// TIA Portal V17 export
// export: Created 2025-03-07T09:17:58.1405762Z, ExportSetting WithDefaults, DisplayName Totally Integrated Automation Portal, DisplayVersion V17 Update 8, DisplayName TIA Portal Openness, DisplayVersion V17 Update 8, DisplayName TIA Portal Version Control Interface, DisplayVersion V17, DisplayName SINAMICS Startdrive Advanced, DisplayVersion V17 SP2, DisplayName SINAMICS Startdrive G110M, G120, G120C, G120D, G120P, G115D, DisplayVersion V17 SP2, DisplayName SINAMICS Startdrive G130, G150, S120, S150, SINAMICS MV, S210, DisplayVersion V17 SP2, DisplayName STEP 7 Professional, DisplayVersion V17 Update 8, DisplayName SINUMERIK ONE STEP 7 Toolbox, DisplayVersion V17 Update 12, DisplayName SINUMERIK 840D sl STEP 7 Toolbox, DisplayVersion V17 Update 12, DisplayName STEP 7 Safety, DisplayVersion V17 Update 6, DisplayName WinCC Advanced, DisplayVersion V17 Update 8
FUNCTION "FC1213_HOME_UNIT_01_STATION_1" : Void   // FC1213, LAD
{ S7_Optimized_Access := 'FALSE' }
AUTHOR : ETXETAR
VERSION : 1.0
// stored: AutoNumber false, IsIECCheckEnabled false, SetENOAutomatically false, UDAEnableTagReadback false
   VAR_TEMP
      UNIT_01_STATION_1_LOCAL_E_RETURNS : Bool;   // UNIT 01 STATION 1 LOCAL E RETURNS
      UNIT_01_STATION_1_MACHINE_E_RETURNS : Bool;   // UNIT 01 STATION 1 MACHINE E RETURNS
   END_VAR
   VAR CONSTANT
      FC_NUMBER : DInt := 1213;
   END_VAR
   VAR_TEMP   // added for the SCL form of the ladder/FBD networks
      _w1 : Bool;
      _w2 : Bool;
   END_VAR
BEGIN

REGION Network 1: GENERAL CONDITIONS
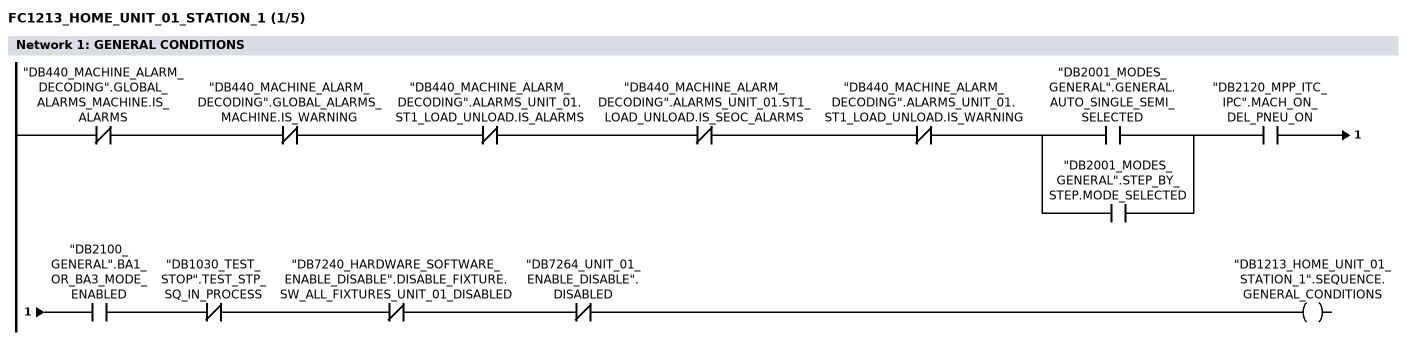
   RUNG wire#powerrail
      I_Contact( "DB440_MACHINE_ALARM_DECODING".GLOBAL_ALARMS_MACHINE.IS_ALARMS )
      I_Contact( "DB440_MACHINE_ALARM_DECODING".GLOBAL_ALARMS_MACHINE.IS_WARNING )
      I_Contact( "DB440_MACHINE_ALARM_DECODING".ALARMS_UNIT_01.ST1_LOAD_UNLOAD.IS_ALARMS )
      I_Contact( "DB440_MACHINE_ALARM_DECODING".ALARMS_UNIT_01.ST1_LOAD_UNLOAD.IS_SEOC_ALARMS )
      I_Contact( "DB440_MACHINE_ALARM_DECODING".ALARMS_UNIT_01.ST1_LOAD_UNLOAD.IS_WARNING )
      wire#w1
      Contact( "DB2001_MODES_GENERAL".GENERAL.AUTO_SINGLE_SEMI_SELECTED )
      wire#w2
      Contact( "DB2120_MPP_ITC_IPC".MACH_ON_DEL_PNEU_ON )
      Contact( "DB2100_GENERAL".BA1_OR_BA3_MODE_ENABLED )
      I_Contact( "DB1030_TEST_STOP".TEST_STP_SQ_IN_PROCESS )
      I_Contact( "DB7240_HARDWARE_SOFTWARE_ENABLE_DISABLE".DISABLE_FIXTURE.SW_ALL_FIXTURES_UNIT_01_DISABLED )
      I_Contact( "DB7264_UNIT_01_ENABLE_DISABLE".DISABLED )
      Coil( "DB1213_HOME_UNIT_01_STATION_1".SEQUENCE.GENERAL_CONDITIONS )
   END_RUNG
   RUNG wire#w1
      Contact( "DB2001_MODES_GENERAL".STEP_BY_STEP.MODE_SELECTED )
   END_RUNG wire#w2
   // the same network as SCL:
   "DB1213_HOME_UNIT_01_STATION_1".SEQUENCE.GENERAL_CONDITIONS := NOT "DB440_MACHINE_ALARM_DECODING".GLOBAL_ALARMS_MACHINE.IS_ALARMS AND NOT "DB440_MACHINE_ALARM_DECODING".GLOBAL_ALARMS_MACHINE.IS_WARNING AND NOT "DB440_MACHINE_ALARM_DECODING".ALARMS_UNIT_01.ST1_LOAD_UNLOAD.IS_ALARMS AND NOT "DB440_MACHINE_ALARM_DECODING".ALARMS_UNIT_01.ST1_LOAD_UNLOAD.IS_SEOC_ALARMS AND NOT "DB440_MACHINE_ALARM_DECODING".ALARMS_UNIT_01.ST1_LOAD_UNLOAD.IS_WARNING AND ("DB2001_MODES_GENERAL".GENERAL.AUTO_SINGLE_SEMI_SELECTED OR "DB2001_MODES_GENERAL".STEP_BY_STEP.MODE_SELECTED) AND "DB2120_MPP_ITC_IPC".MACH_ON_DEL_PNEU_ON AND "DB2100_GENERAL".BA1_OR_BA3_MODE_ENABLED AND NOT "DB1030_TEST_STOP".TEST_STP_SQ_IN_PROCESS AND NOT "DB7240_HARDWARE_SOFTWARE_ENABLE_DISABLE".DISABLE_FIXTURE.SW_ALL_FIXTURES_UNIT_01_DISABLED AND NOT "DB7264_UNIT_01_ENABLE_DISABLE".DISABLED;
END_REGION

REGION Network 2: OPERATOR HELP
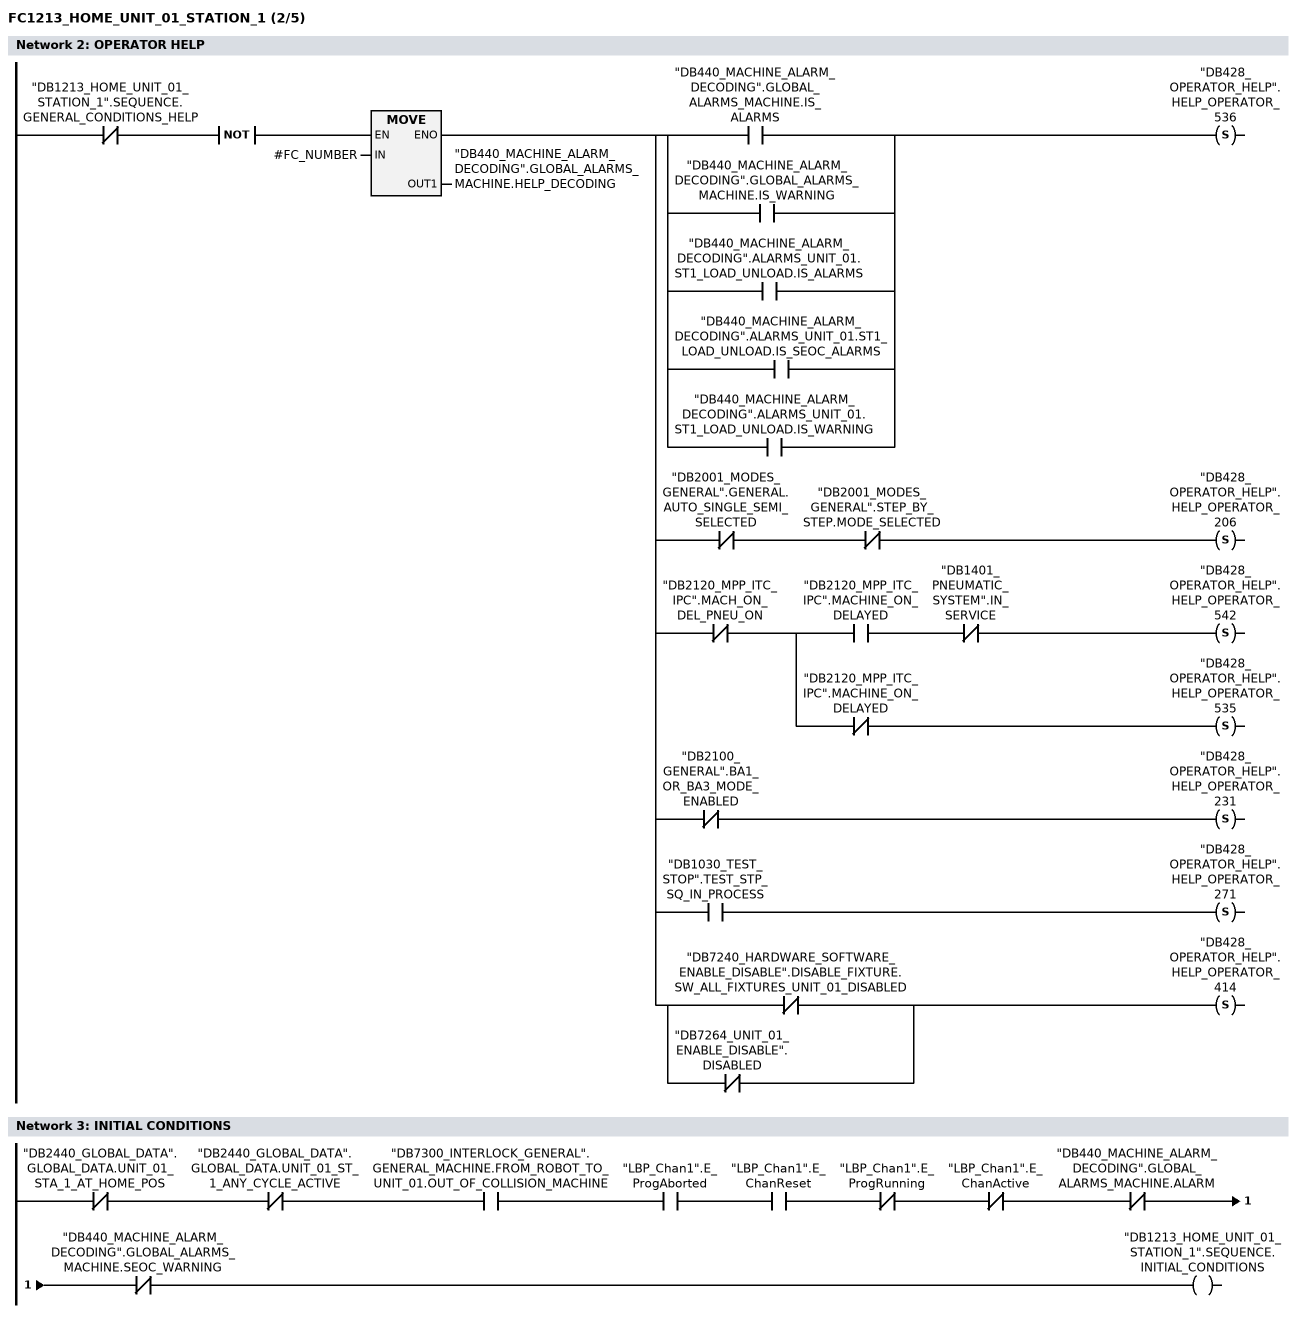
   RUNG wire#powerrail
      I_Contact( "DB1213_HOME_UNIT_01_STATION_1".SEQUENCE.GENERAL_CONDITIONS_HELP )
      Not()
      { S7_GenerateENO := "TRUE" } Move(in := #FC_NUMBER, out1 => "DB440_MACHINE_ALARM_DECODING".GLOBAL_ALARMS_MACHINE.HELP_DECODING)
      wire#w1
      Contact( "DB440_MACHINE_ALARM_DECODING".GLOBAL_ALARMS_MACHINE.IS_ALARMS )
      wire#w2
      S_Coil( "DB428_OPERATOR_HELP".HELP_OPERATOR_536 )
   END_RUNG
   RUNG wire#w1
      Contact( "DB440_MACHINE_ALARM_DECODING".GLOBAL_ALARMS_MACHINE.IS_WARNING )
   END_RUNG wire#w2
   RUNG wire#w1
      Contact( "DB440_MACHINE_ALARM_DECODING".ALARMS_UNIT_01.ST1_LOAD_UNLOAD.IS_ALARMS )
   END_RUNG wire#w2
   RUNG wire#w1
      Contact( "DB440_MACHINE_ALARM_DECODING".ALARMS_UNIT_01.ST1_LOAD_UNLOAD.IS_SEOC_ALARMS )
   END_RUNG wire#w2
   RUNG wire#w1
      Contact( "DB440_MACHINE_ALARM_DECODING".ALARMS_UNIT_01.ST1_LOAD_UNLOAD.IS_WARNING )
   END_RUNG wire#w2
   RUNG wire#w1
      I_Contact( "DB2001_MODES_GENERAL".GENERAL.AUTO_SINGLE_SEMI_SELECTED )
      I_Contact( "DB2001_MODES_GENERAL".STEP_BY_STEP.MODE_SELECTED )
      S_Coil( "DB428_OPERATOR_HELP".HELP_OPERATOR_206 )
   END_RUNG
   RUNG wire#w1
      I_Contact( "DB2120_MPP_ITC_IPC".MACH_ON_DEL_PNEU_ON )
      wire#w3
      Contact( "DB2120_MPP_ITC_IPC".MACHINE_ON_DELAYED )
      I_Contact( "DB1401_PNEUMATIC_SYSTEM".IN_SERVICE )
      S_Coil( "DB428_OPERATOR_HELP".HELP_OPERATOR_542 )
   END_RUNG
   RUNG wire#w3
      I_Contact( "DB2120_MPP_ITC_IPC".MACHINE_ON_DELAYED )
      S_Coil( "DB428_OPERATOR_HELP".HELP_OPERATOR_535 )
   END_RUNG
   RUNG wire#w1
      I_Contact( "DB2100_GENERAL".BA1_OR_BA3_MODE_ENABLED )
      S_Coil( "DB428_OPERATOR_HELP".HELP_OPERATOR_231 )
   END_RUNG
   RUNG wire#w1
      Contact( "DB1030_TEST_STOP".TEST_STP_SQ_IN_PROCESS )
      S_Coil( "DB428_OPERATOR_HELP".HELP_OPERATOR_271 )
   END_RUNG
   RUNG wire#w1
      I_Contact( "DB7240_HARDWARE_SOFTWARE_ENABLE_DISABLE".DISABLE_FIXTURE.SW_ALL_FIXTURES_UNIT_01_DISABLED )
      wire#w4
      S_Coil( "DB428_OPERATOR_HELP".HELP_OPERATOR_414 )
   END_RUNG
   RUNG wire#w1
      I_Contact( "DB7264_UNIT_01_ENABLE_DISABLE".DISABLED )
   END_RUNG wire#w4
   // the same network as SCL:
   // ENO of a box is taken as its EN; it also drops when the box reports an error
   #_w1 := NOT (NOT "DB1213_HOME_UNIT_01_STATION_1".SEQUENCE.GENERAL_CONDITIONS_HELP);
   IF #_w1 THEN "DB440_MACHINE_ALARM_DECODING".GLOBAL_ALARMS_MACHINE.HELP_DECODING := #FC_NUMBER; END_IF;
   IF #_w1 AND ("DB440_MACHINE_ALARM_DECODING".GLOBAL_ALARMS_MACHINE.IS_ALARMS OR "DB440_MACHINE_ALARM_DECODING".GLOBAL_ALARMS_MACHINE.IS_WARNING OR "DB440_MACHINE_ALARM_DECODING".ALARMS_UNIT_01.ST1_LOAD_UNLOAD.IS_ALARMS OR "DB440_MACHINE_ALARM_DECODING".ALARMS_UNIT_01.ST1_LOAD_UNLOAD.IS_SEOC_ALARMS OR "DB440_MACHINE_ALARM_DECODING".ALARMS_UNIT_01.ST1_LOAD_UNLOAD.IS_WARNING) THEN
       "DB428_OPERATOR_HELP".HELP_OPERATOR_536 := TRUE;
   END_IF;
   IF #_w1 AND NOT "DB2001_MODES_GENERAL".GENERAL.AUTO_SINGLE_SEMI_SELECTED AND NOT "DB2001_MODES_GENERAL".STEP_BY_STEP.MODE_SELECTED THEN
       "DB428_OPERATOR_HELP".HELP_OPERATOR_206 := TRUE;
   END_IF;
   #_w2 := #_w1 AND NOT "DB2120_MPP_ITC_IPC".MACH_ON_DEL_PNEU_ON;
   IF #_w2 AND "DB2120_MPP_ITC_IPC".MACHINE_ON_DELAYED AND NOT "DB1401_PNEUMATIC_SYSTEM".IN_SERVICE THEN
       "DB428_OPERATOR_HELP".HELP_OPERATOR_542 := TRUE;
   END_IF;
   IF #_w2 AND NOT "DB2120_MPP_ITC_IPC".MACHINE_ON_DELAYED THEN
       "DB428_OPERATOR_HELP".HELP_OPERATOR_535 := TRUE;
   END_IF;
   IF #_w1 AND NOT "DB2100_GENERAL".BA1_OR_BA3_MODE_ENABLED THEN
       "DB428_OPERATOR_HELP".HELP_OPERATOR_231 := TRUE;
   END_IF;
   IF #_w1 AND "DB1030_TEST_STOP".TEST_STP_SQ_IN_PROCESS THEN
       "DB428_OPERATOR_HELP".HELP_OPERATOR_271 := TRUE;
   END_IF;
   IF #_w1 AND (NOT "DB7240_HARDWARE_SOFTWARE_ENABLE_DISABLE".DISABLE_FIXTURE.SW_ALL_FIXTURES_UNIT_01_DISABLED OR NOT "DB7264_UNIT_01_ENABLE_DISABLE".DISABLED) THEN
       "DB428_OPERATOR_HELP".HELP_OPERATOR_414 := TRUE;
   END_IF;
END_REGION

REGION Network 3: INITIAL CONDITIONS
   RUNG wire#powerrail
      I_Contact( "DB2440_GLOBAL_DATA".GLOBAL_DATA.UNIT_01_STA_1_AT_HOME_POS )
      I_Contact( "DB2440_GLOBAL_DATA".GLOBAL_DATA.UNIT_01_ST_1_ANY_CYCLE_ACTIVE )
      Contact( "DB7300_INTERLOCK_GENERAL".GENERAL_MACHINE.FROM_ROBOT_TO_UNIT_01.OUT_OF_COLLISION_MACHINE )
      Contact( "LBP_Chan1".E_ProgAborted )
      Contact( "LBP_Chan1".E_ChanReset )
      I_Contact( "LBP_Chan1".E_ProgRunning )
      I_Contact( "LBP_Chan1".E_ChanActive )
      I_Contact( "DB440_MACHINE_ALARM_DECODING".GLOBAL_ALARMS_MACHINE.ALARM )
      I_Contact( "DB440_MACHINE_ALARM_DECODING".GLOBAL_ALARMS_MACHINE.SEOC_WARNING )
      Coil( "DB1213_HOME_UNIT_01_STATION_1".SEQUENCE.INITIAL_CONDITIONS )
   END_RUNG
   // the same network as SCL:
   "DB1213_HOME_UNIT_01_STATION_1".SEQUENCE.INITIAL_CONDITIONS := NOT "DB2440_GLOBAL_DATA".GLOBAL_DATA.UNIT_01_STA_1_AT_HOME_POS AND NOT "DB2440_GLOBAL_DATA".GLOBAL_DATA.UNIT_01_ST_1_ANY_CYCLE_ACTIVE AND "DB7300_INTERLOCK_GENERAL".GENERAL_MACHINE.FROM_ROBOT_TO_UNIT_01.OUT_OF_COLLISION_MACHINE AND "LBP_Chan1".E_ProgAborted AND "LBP_Chan1".E_ChanReset AND NOT "LBP_Chan1".E_ProgRunning AND NOT "LBP_Chan1".E_ChanActive AND NOT "DB440_MACHINE_ALARM_DECODING".GLOBAL_ALARMS_MACHINE.ALARM AND NOT "DB440_MACHINE_ALARM_DECODING".GLOBAL_ALARMS_MACHINE.SEOC_WARNING;
END_REGION

REGION Network 4: OPERATOR HELP
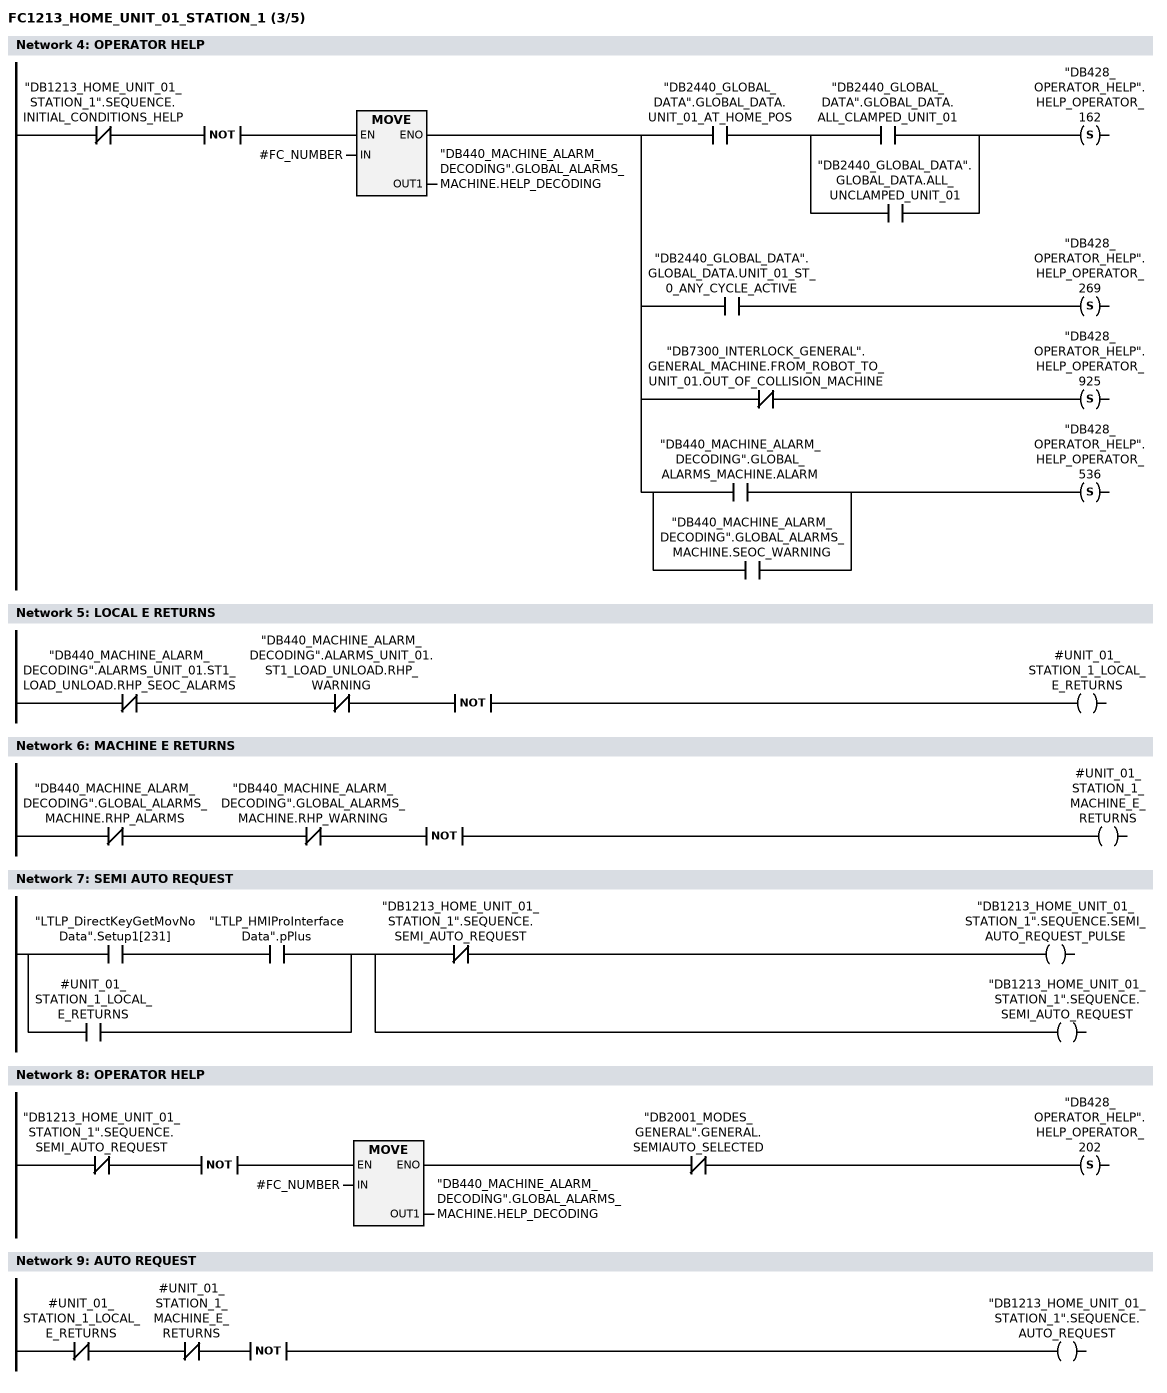
   RUNG wire#powerrail
      I_Contact( "DB1213_HOME_UNIT_01_STATION_1".SEQUENCE.INITIAL_CONDITIONS_HELP )
      Not()
      { S7_GenerateENO := "TRUE" } Move(in := #FC_NUMBER, out1 => "DB440_MACHINE_ALARM_DECODING".GLOBAL_ALARMS_MACHINE.HELP_DECODING)
      wire#w1
      Contact( "DB2440_GLOBAL_DATA".GLOBAL_DATA.UNIT_01_AT_HOME_POS )
      wire#w2
      Contact( "DB2440_GLOBAL_DATA".GLOBAL_DATA.ALL_CLAMPED_UNIT_01 )
      wire#w3
      S_Coil( "DB428_OPERATOR_HELP".HELP_OPERATOR_162 )
   END_RUNG
   RUNG wire#w2
      Contact( "DB2440_GLOBAL_DATA".GLOBAL_DATA.ALL_UNCLAMPED_UNIT_01 )
   END_RUNG wire#w3
   RUNG wire#w1
      Contact( "DB2440_GLOBAL_DATA".GLOBAL_DATA.UNIT_01_ST_0_ANY_CYCLE_ACTIVE )
      S_Coil( "DB428_OPERATOR_HELP".HELP_OPERATOR_269 )
   END_RUNG
   RUNG wire#w1
      I_Contact( "DB7300_INTERLOCK_GENERAL".GENERAL_MACHINE.FROM_ROBOT_TO_UNIT_01.OUT_OF_COLLISION_MACHINE )
      S_Coil( "DB428_OPERATOR_HELP".HELP_OPERATOR_925 )
   END_RUNG
   RUNG wire#w1
      Contact( "DB440_MACHINE_ALARM_DECODING".GLOBAL_ALARMS_MACHINE.ALARM )
      wire#w4
      S_Coil( "DB428_OPERATOR_HELP".HELP_OPERATOR_536 )
   END_RUNG
   RUNG wire#w1
      Contact( "DB440_MACHINE_ALARM_DECODING".GLOBAL_ALARMS_MACHINE.SEOC_WARNING )
   END_RUNG wire#w4
   // the same network as SCL:
   // ENO of a box is taken as its EN; it also drops when the box reports an error
   #_w1 := NOT (NOT "DB1213_HOME_UNIT_01_STATION_1".SEQUENCE.INITIAL_CONDITIONS_HELP);
   IF #_w1 THEN "DB440_MACHINE_ALARM_DECODING".GLOBAL_ALARMS_MACHINE.HELP_DECODING := #FC_NUMBER; END_IF;
   IF #_w1 AND "DB2440_GLOBAL_DATA".GLOBAL_DATA.UNIT_01_AT_HOME_POS AND ("DB2440_GLOBAL_DATA".GLOBAL_DATA.ALL_CLAMPED_UNIT_01 OR "DB2440_GLOBAL_DATA".GLOBAL_DATA.ALL_UNCLAMPED_UNIT_01) THEN
       "DB428_OPERATOR_HELP".HELP_OPERATOR_162 := TRUE;
   END_IF;
   IF #_w1 AND "DB2440_GLOBAL_DATA".GLOBAL_DATA.UNIT_01_ST_0_ANY_CYCLE_ACTIVE THEN
       "DB428_OPERATOR_HELP".HELP_OPERATOR_269 := TRUE;
   END_IF;
   IF #_w1 AND NOT "DB7300_INTERLOCK_GENERAL".GENERAL_MACHINE.FROM_ROBOT_TO_UNIT_01.OUT_OF_COLLISION_MACHINE THEN
       "DB428_OPERATOR_HELP".HELP_OPERATOR_925 := TRUE;
   END_IF;
   IF #_w1 AND ("DB440_MACHINE_ALARM_DECODING".GLOBAL_ALARMS_MACHINE.ALARM OR "DB440_MACHINE_ALARM_DECODING".GLOBAL_ALARMS_MACHINE.SEOC_WARNING) THEN
       "DB428_OPERATOR_HELP".HELP_OPERATOR_536 := TRUE;
   END_IF;
END_REGION

REGION Network 5: LOCAL E RETURNS
   RUNG wire#powerrail
      I_Contact( "DB440_MACHINE_ALARM_DECODING".ALARMS_UNIT_01.ST1_LOAD_UNLOAD.RHP_SEOC_ALARMS )
      I_Contact( "DB440_MACHINE_ALARM_DECODING".ALARMS_UNIT_01.ST1_LOAD_UNLOAD.RHP_WARNING )
      Not()
      Coil( #UNIT_01_STATION_1_LOCAL_E_RETURNS )
   END_RUNG
   // the same network as SCL:
   #UNIT_01_STATION_1_LOCAL_E_RETURNS := NOT (NOT "DB440_MACHINE_ALARM_DECODING".ALARMS_UNIT_01.ST1_LOAD_UNLOAD.RHP_SEOC_ALARMS AND NOT "DB440_MACHINE_ALARM_DECODING".ALARMS_UNIT_01.ST1_LOAD_UNLOAD.RHP_WARNING);
END_REGION

REGION Network 6: MACHINE E RETURNS
   RUNG wire#powerrail
      I_Contact( "DB440_MACHINE_ALARM_DECODING".GLOBAL_ALARMS_MACHINE.RHP_ALARMS )
      I_Contact( "DB440_MACHINE_ALARM_DECODING".GLOBAL_ALARMS_MACHINE.RHP_WARNING )
      Not()
      Coil( #UNIT_01_STATION_1_MACHINE_E_RETURNS )
   END_RUNG
   // the same network as SCL:
   #UNIT_01_STATION_1_MACHINE_E_RETURNS := NOT (NOT "DB440_MACHINE_ALARM_DECODING".GLOBAL_ALARMS_MACHINE.RHP_ALARMS AND NOT "DB440_MACHINE_ALARM_DECODING".GLOBAL_ALARMS_MACHINE.RHP_WARNING);
END_REGION

REGION Network 7: SEMI AUTO REQUEST
   RUNG wire#powerrail
      Contact( "LTLP_DirectKeyGetMovNoData".Setup1[231] )
      Contact( "LTLP_HMIProInterfaceData".pPlus )
      wire#w1
      I_Contact( "DB1213_HOME_UNIT_01_STATION_1".SEQUENCE.SEMI_AUTO_REQUEST )
      Coil( "DB1213_HOME_UNIT_01_STATION_1".SEQUENCE.SEMI_AUTO_REQUEST_PULSE )
   END_RUNG
   RUNG wire#powerrail
      Contact( #UNIT_01_STATION_1_LOCAL_E_RETURNS )
   END_RUNG wire#w1
   RUNG wire#w1
      Coil( "DB1213_HOME_UNIT_01_STATION_1".SEQUENCE.SEMI_AUTO_REQUEST )
   END_RUNG
   // the same network as SCL:
   #_w1 := ("LTLP_DirectKeyGetMovNoData".Setup1[231] AND "LTLP_HMIProInterfaceData".pPlus) OR #UNIT_01_STATION_1_LOCAL_E_RETURNS;
   "DB1213_HOME_UNIT_01_STATION_1".SEQUENCE.SEMI_AUTO_REQUEST_PULSE := #_w1 AND NOT "DB1213_HOME_UNIT_01_STATION_1".SEQUENCE.SEMI_AUTO_REQUEST;
   "DB1213_HOME_UNIT_01_STATION_1".SEQUENCE.SEMI_AUTO_REQUEST := #_w1;
END_REGION

REGION Network 8: OPERATOR HELP
   RUNG wire#powerrail
      I_Contact( "DB1213_HOME_UNIT_01_STATION_1".SEQUENCE.SEMI_AUTO_REQUEST )
      Not()
      { S7_GenerateENO := "TRUE" } Move(in := #FC_NUMBER, out1 => "DB440_MACHINE_ALARM_DECODING".GLOBAL_ALARMS_MACHINE.HELP_DECODING)
      I_Contact( "DB2001_MODES_GENERAL".GENERAL.SEMIAUTO_SELECTED )
      S_Coil( "DB428_OPERATOR_HELP".HELP_OPERATOR_202 )
   END_RUNG
   // the same network as SCL:
   // ENO of a box is taken as its EN; it also drops when the box reports an error
   #_w1 := NOT (NOT "DB1213_HOME_UNIT_01_STATION_1".SEQUENCE.SEMI_AUTO_REQUEST);
   IF #_w1 THEN "DB440_MACHINE_ALARM_DECODING".GLOBAL_ALARMS_MACHINE.HELP_DECODING := #FC_NUMBER; END_IF;
   IF #_w1 AND NOT "DB2001_MODES_GENERAL".GENERAL.SEMIAUTO_SELECTED THEN
       "DB428_OPERATOR_HELP".HELP_OPERATOR_202 := TRUE;
   END_IF;
END_REGION

REGION Network 9: AUTO REQUEST
   RUNG wire#powerrail
      I_Contact( #UNIT_01_STATION_1_LOCAL_E_RETURNS )
      I_Contact( #UNIT_01_STATION_1_MACHINE_E_RETURNS )
      Not()
      Coil( "DB1213_HOME_UNIT_01_STATION_1".SEQUENCE.AUTO_REQUEST )
   END_RUNG
   // the same network as SCL:
   "DB1213_HOME_UNIT_01_STATION_1".SEQUENCE.AUTO_REQUEST := NOT (NOT #UNIT_01_STATION_1_LOCAL_E_RETURNS AND NOT #UNIT_01_STATION_1_MACHINE_E_RETURNS);
END_REGION

REGION Network 10: REQUEST
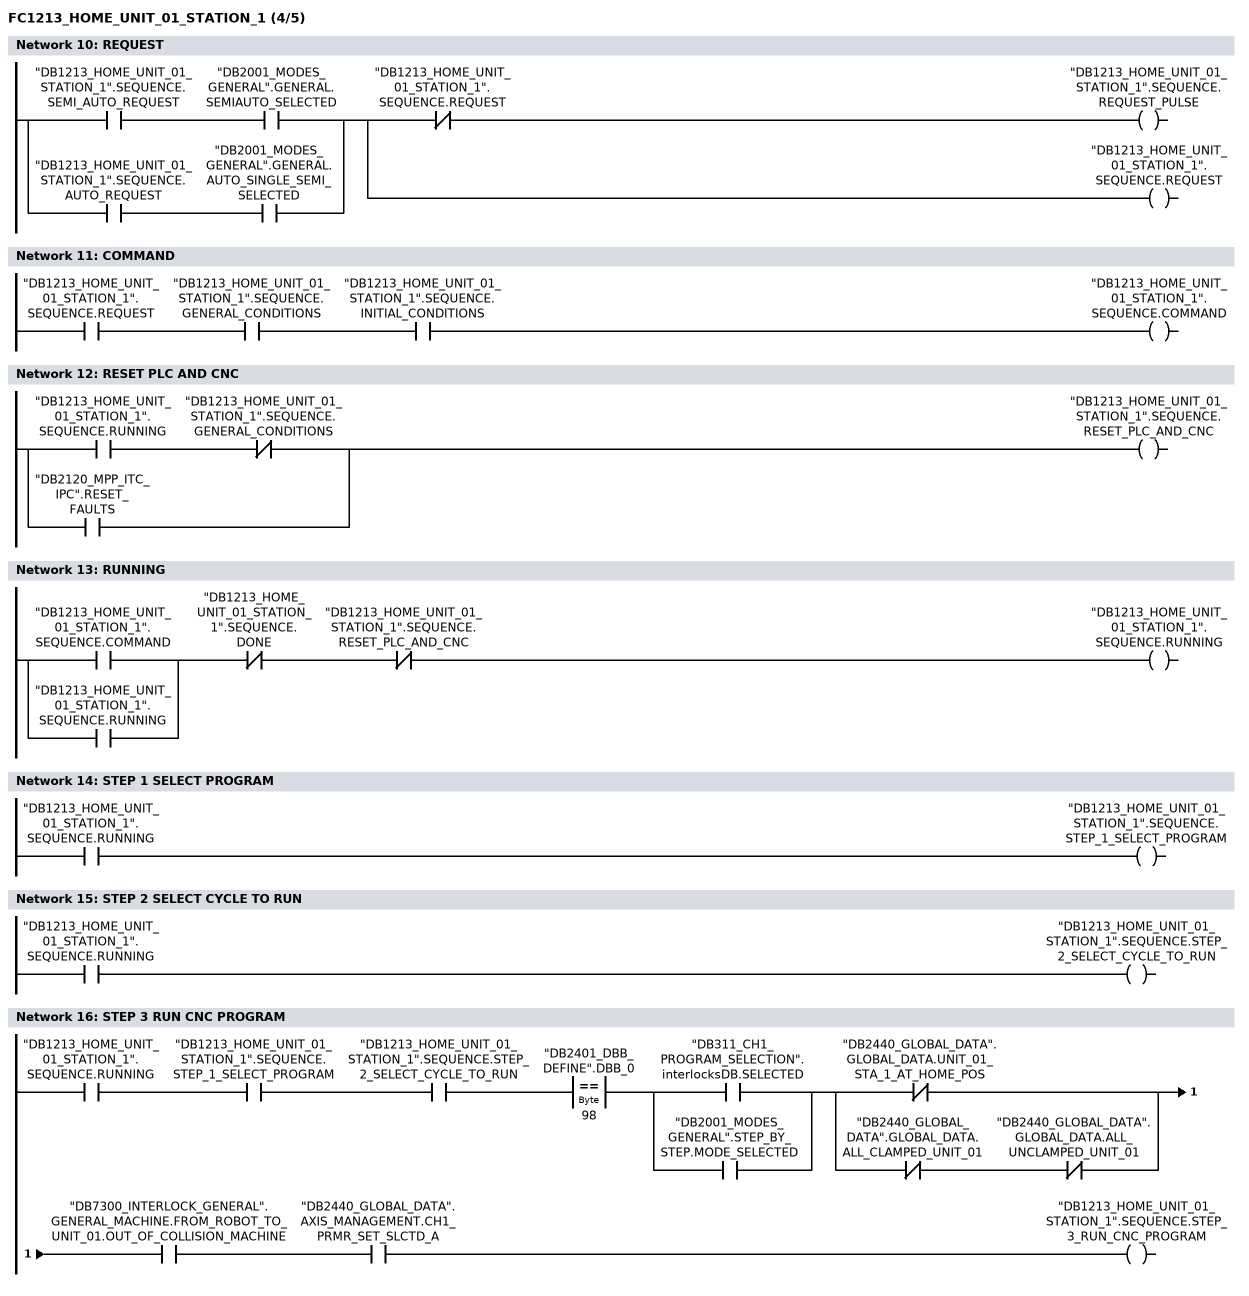
   RUNG wire#powerrail
      Contact( "DB1213_HOME_UNIT_01_STATION_1".SEQUENCE.SEMI_AUTO_REQUEST )
      Contact( "DB2001_MODES_GENERAL".GENERAL.SEMIAUTO_SELECTED )
      wire#w1
      I_Contact( "DB1213_HOME_UNIT_01_STATION_1".SEQUENCE.REQUEST )
      Coil( "DB1213_HOME_UNIT_01_STATION_1".SEQUENCE.REQUEST_PULSE )
   END_RUNG
   RUNG wire#powerrail
      Contact( "DB1213_HOME_UNIT_01_STATION_1".SEQUENCE.AUTO_REQUEST )
      Contact( "DB2001_MODES_GENERAL".GENERAL.AUTO_SINGLE_SEMI_SELECTED )
   END_RUNG wire#w1
   RUNG wire#w1
      Coil( "DB1213_HOME_UNIT_01_STATION_1".SEQUENCE.REQUEST )
   END_RUNG
   // the same network as SCL:
   #_w1 := ("DB1213_HOME_UNIT_01_STATION_1".SEQUENCE.SEMI_AUTO_REQUEST AND "DB2001_MODES_GENERAL".GENERAL.SEMIAUTO_SELECTED) OR ("DB1213_HOME_UNIT_01_STATION_1".SEQUENCE.AUTO_REQUEST AND "DB2001_MODES_GENERAL".GENERAL.AUTO_SINGLE_SEMI_SELECTED);
   "DB1213_HOME_UNIT_01_STATION_1".SEQUENCE.REQUEST_PULSE := #_w1 AND NOT "DB1213_HOME_UNIT_01_STATION_1".SEQUENCE.REQUEST;
   "DB1213_HOME_UNIT_01_STATION_1".SEQUENCE.REQUEST := #_w1;
END_REGION

REGION Network 11: COMMAND
   RUNG wire#powerrail
      Contact( "DB1213_HOME_UNIT_01_STATION_1".SEQUENCE.REQUEST )
      Contact( "DB1213_HOME_UNIT_01_STATION_1".SEQUENCE.GENERAL_CONDITIONS )
      Contact( "DB1213_HOME_UNIT_01_STATION_1".SEQUENCE.INITIAL_CONDITIONS )
      Coil( "DB1213_HOME_UNIT_01_STATION_1".SEQUENCE.COMMAND )
   END_RUNG
   // the same network as SCL:
   "DB1213_HOME_UNIT_01_STATION_1".SEQUENCE.COMMAND := "DB1213_HOME_UNIT_01_STATION_1".SEQUENCE.REQUEST AND "DB1213_HOME_UNIT_01_STATION_1".SEQUENCE.GENERAL_CONDITIONS AND "DB1213_HOME_UNIT_01_STATION_1".SEQUENCE.INITIAL_CONDITIONS;
END_REGION

REGION Network 12: RESET PLC AND CNC
   RUNG wire#powerrail
      Contact( "DB1213_HOME_UNIT_01_STATION_1".SEQUENCE.RUNNING )
      I_Contact( "DB1213_HOME_UNIT_01_STATION_1".SEQUENCE.GENERAL_CONDITIONS )
      wire#w1
      Coil( "DB1213_HOME_UNIT_01_STATION_1".SEQUENCE.RESET_PLC_AND_CNC )
   END_RUNG
   RUNG wire#powerrail
      Contact( "DB2120_MPP_ITC_IPC".RESET_FAULTS )
   END_RUNG wire#w1
   // the same network as SCL:
   "DB1213_HOME_UNIT_01_STATION_1".SEQUENCE.RESET_PLC_AND_CNC := ("DB1213_HOME_UNIT_01_STATION_1".SEQUENCE.RUNNING AND NOT "DB1213_HOME_UNIT_01_STATION_1".SEQUENCE.GENERAL_CONDITIONS) OR "DB2120_MPP_ITC_IPC".RESET_FAULTS;
END_REGION

REGION Network 13: RUNNING
   RUNG wire#powerrail
      Contact( "DB1213_HOME_UNIT_01_STATION_1".SEQUENCE.COMMAND )
      wire#w1
      I_Contact( "DB1213_HOME_UNIT_01_STATION_1".SEQUENCE.DONE )
      I_Contact( "DB1213_HOME_UNIT_01_STATION_1".SEQUENCE.RESET_PLC_AND_CNC )
      Coil( "DB1213_HOME_UNIT_01_STATION_1".SEQUENCE.RUNNING )
   END_RUNG
   RUNG wire#powerrail
      Contact( "DB1213_HOME_UNIT_01_STATION_1".SEQUENCE.RUNNING )
   END_RUNG wire#w1
   // the same network as SCL:
   "DB1213_HOME_UNIT_01_STATION_1".SEQUENCE.RUNNING := ("DB1213_HOME_UNIT_01_STATION_1".SEQUENCE.COMMAND OR "DB1213_HOME_UNIT_01_STATION_1".SEQUENCE.RUNNING) AND NOT "DB1213_HOME_UNIT_01_STATION_1".SEQUENCE.DONE AND NOT "DB1213_HOME_UNIT_01_STATION_1".SEQUENCE.RESET_PLC_AND_CNC;
END_REGION

REGION Network 14: STEP 1 SELECT PROGRAM
   RUNG wire#powerrail
      Contact( "DB1213_HOME_UNIT_01_STATION_1".SEQUENCE.RUNNING )
      Coil( "DB1213_HOME_UNIT_01_STATION_1".SEQUENCE.STEP_1_SELECT_PROGRAM )
   END_RUNG
   // the same network as SCL:
   "DB1213_HOME_UNIT_01_STATION_1".SEQUENCE.STEP_1_SELECT_PROGRAM := "DB1213_HOME_UNIT_01_STATION_1".SEQUENCE.RUNNING;
END_REGION

REGION Network 15: STEP 2 SELECT CYCLE TO RUN
   RUNG wire#powerrail
      Contact( "DB1213_HOME_UNIT_01_STATION_1".SEQUENCE.RUNNING )
      Coil( "DB1213_HOME_UNIT_01_STATION_1".SEQUENCE.STEP_2_SELECT_CYCLE_TO_RUN )
   END_RUNG
   // the same network as SCL:
   "DB1213_HOME_UNIT_01_STATION_1".SEQUENCE.STEP_2_SELECT_CYCLE_TO_RUN := "DB1213_HOME_UNIT_01_STATION_1".SEQUENCE.RUNNING;
END_REGION

REGION Network 16: STEP 3 RUN CNC PROGRAM
   RUNG wire#powerrail
      Contact( "DB1213_HOME_UNIT_01_STATION_1".SEQUENCE.RUNNING )
      Contact( "DB1213_HOME_UNIT_01_STATION_1".SEQUENCE.STEP_1_SELECT_PROGRAM )
      Contact( "DB1213_HOME_UNIT_01_STATION_1".SEQUENCE.STEP_2_SELECT_CYCLE_TO_RUN )
      { S7_Templates := "SrcType := Byte" } EQ_Contact(in1 := "DB2401_DBB_DEFINE".DBB_0, in2 := 98)
      wire#w1
      Contact( "DB311_CH1_PROGRAM_SELECTION".interlocksDB.SELECTED )
      wire#w2
      I_Contact( "DB2440_GLOBAL_DATA".GLOBAL_DATA.UNIT_01_STA_1_AT_HOME_POS )
      wire#w3
      Contact( "DB7300_INTERLOCK_GENERAL".GENERAL_MACHINE.FROM_ROBOT_TO_UNIT_01.OUT_OF_COLLISION_MACHINE )
      Contact( "DB2440_GLOBAL_DATA".AXIS_MANAGEMENT.CH1_PRMR_SET_SLCTD_A )
      Coil( "DB1213_HOME_UNIT_01_STATION_1".SEQUENCE.STEP_3_RUN_CNC_PROGRAM )
   END_RUNG
   RUNG wire#w1
      Contact( "DB2001_MODES_GENERAL".STEP_BY_STEP.MODE_SELECTED )
   END_RUNG wire#w2
   RUNG wire#w2
      I_Contact( "DB2440_GLOBAL_DATA".GLOBAL_DATA.ALL_CLAMPED_UNIT_01 )
      I_Contact( "DB2440_GLOBAL_DATA".GLOBAL_DATA.ALL_UNCLAMPED_UNIT_01 )
   END_RUNG wire#w3
   // the same network as SCL:
   "DB1213_HOME_UNIT_01_STATION_1".SEQUENCE.STEP_3_RUN_CNC_PROGRAM := "DB1213_HOME_UNIT_01_STATION_1".SEQUENCE.RUNNING AND "DB1213_HOME_UNIT_01_STATION_1".SEQUENCE.STEP_1_SELECT_PROGRAM AND "DB1213_HOME_UNIT_01_STATION_1".SEQUENCE.STEP_2_SELECT_CYCLE_TO_RUN AND ("DB2401_DBB_DEFINE".DBB_0 = 98) AND ("DB311_CH1_PROGRAM_SELECTION".interlocksDB.SELECTED OR "DB2001_MODES_GENERAL".STEP_BY_STEP.MODE_SELECTED) AND (NOT "DB2440_GLOBAL_DATA".GLOBAL_DATA.UNIT_01_STA_1_AT_HOME_POS OR (NOT "DB2440_GLOBAL_DATA".GLOBAL_DATA.ALL_CLAMPED_UNIT_01 AND NOT "DB2440_GLOBAL_DATA".GLOBAL_DATA.ALL_UNCLAMPED_UNIT_01)) AND "DB7300_INTERLOCK_GENERAL".GENERAL_MACHINE.FROM_ROBOT_TO_UNIT_01.OUT_OF_COLLISION_MACHINE AND "DB2440_GLOBAL_DATA".AXIS_MANAGEMENT.CH1_PRMR_SET_SLCTD_A;
END_REGION

REGION Network 17: DONE
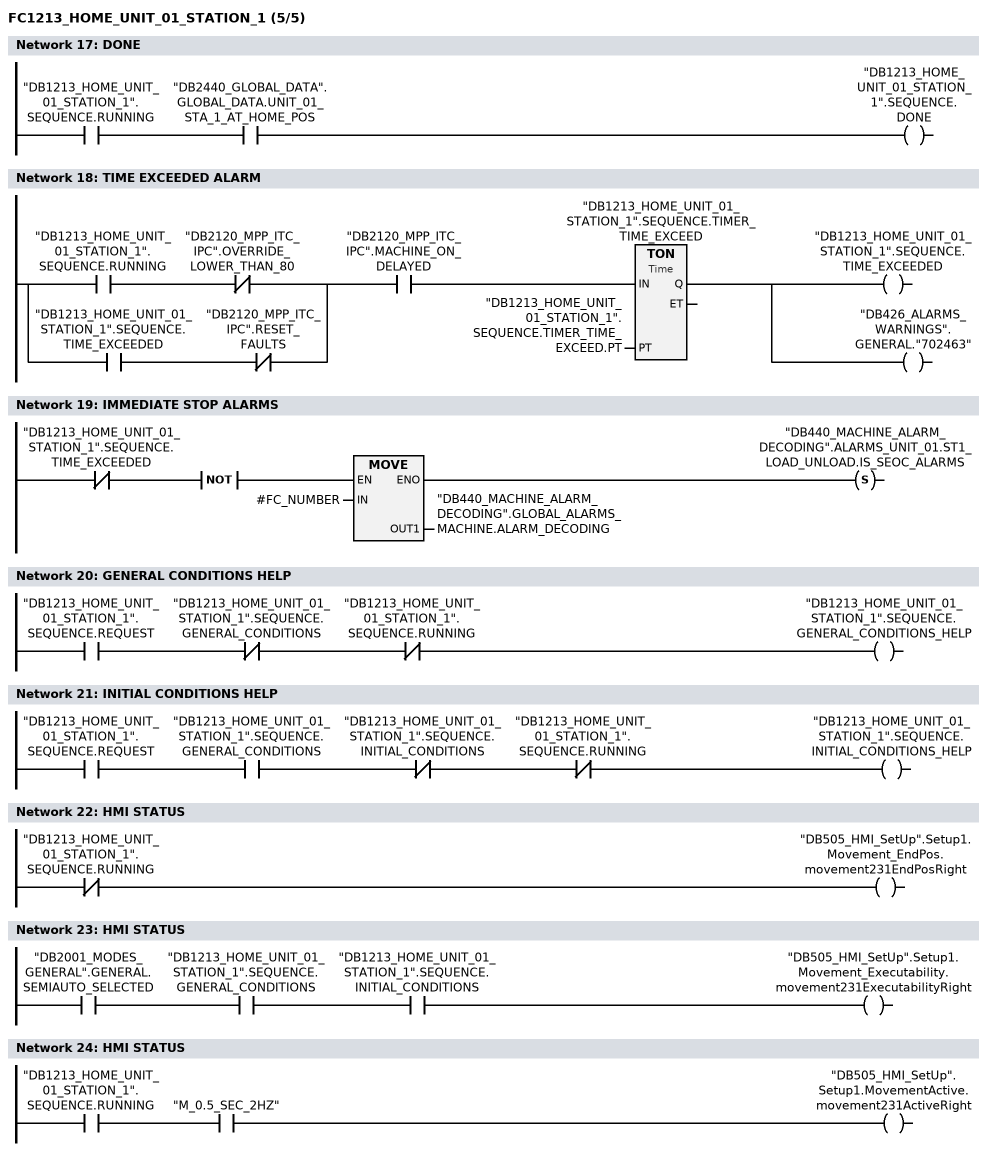
   RUNG wire#powerrail
      Contact( "DB1213_HOME_UNIT_01_STATION_1".SEQUENCE.RUNNING )
      Contact( "DB2440_GLOBAL_DATA".GLOBAL_DATA.UNIT_01_STA_1_AT_HOME_POS )
      Coil( "DB1213_HOME_UNIT_01_STATION_1".SEQUENCE.DONE )
   END_RUNG
   // the same network as SCL:
   "DB1213_HOME_UNIT_01_STATION_1".SEQUENCE.DONE := "DB1213_HOME_UNIT_01_STATION_1".SEQUENCE.RUNNING AND "DB2440_GLOBAL_DATA".GLOBAL_DATA.UNIT_01_STA_1_AT_HOME_POS;
END_REGION

REGION Network 18: TIME EXCEEDED ALARM
   RUNG wire#powerrail
      Contact( "DB1213_HOME_UNIT_01_STATION_1".SEQUENCE.RUNNING )
      I_Contact( "DB2120_MPP_ITC_IPC".OVERRIDE_LOWER_THAN_80 )
      wire#w1
      Contact( "DB2120_MPP_ITC_IPC".MACHINE_ON_DELAYED )
      { S7_Templates := "time_type := Time" } "DB1213_HOME_UNIT_01_STATION_1".SEQUENCE.TIMER_TIME_EXCEED.TON(pt := "DB1213_HOME_UNIT_01_STATION_1".SEQUENCE.TIMER_TIME_EXCEED.PT, et =>)
      wire#w2
      Coil( "DB1213_HOME_UNIT_01_STATION_1".SEQUENCE.TIME_EXCEEDED )
   END_RUNG
   RUNG wire#powerrail
      Contact( "DB1213_HOME_UNIT_01_STATION_1".SEQUENCE.TIME_EXCEEDED )
      I_Contact( "DB2120_MPP_ITC_IPC".RESET_FAULTS )
   END_RUNG wire#w1
   RUNG wire#w2
      Coil( "DB426_ALARMS_WARNINGS".GENERAL."702463" )
   END_RUNG
   // the same network as SCL:
   "DB1213_HOME_UNIT_01_STATION_1".SEQUENCE.TIMER_TIME_EXCEED.TON(IN := (("DB1213_HOME_UNIT_01_STATION_1".SEQUENCE.RUNNING AND NOT "DB2120_MPP_ITC_IPC".OVERRIDE_LOWER_THAN_80) OR ("DB1213_HOME_UNIT_01_STATION_1".SEQUENCE.TIME_EXCEEDED AND NOT "DB2120_MPP_ITC_IPC".RESET_FAULTS)) AND "DB2120_MPP_ITC_IPC".MACHINE_ON_DELAYED,
                           PT := "DB1213_HOME_UNIT_01_STATION_1".SEQUENCE.TIMER_TIME_EXCEED.PT);
   "DB1213_HOME_UNIT_01_STATION_1".SEQUENCE.TIME_EXCEEDED := "DB1213_HOME_UNIT_01_STATION_1".SEQUENCE.TIMER_TIME_EXCEED.Q;
   "DB426_ALARMS_WARNINGS".GENERAL."702463" := "DB1213_HOME_UNIT_01_STATION_1".SEQUENCE.TIMER_TIME_EXCEED.Q;
END_REGION

REGION Network 19: IMMEDIATE STOP ALARMS
   RUNG wire#powerrail
      I_Contact( "DB1213_HOME_UNIT_01_STATION_1".SEQUENCE.TIME_EXCEEDED )
      Not()
      { S7_GenerateENO := "TRUE" } Move(in := #FC_NUMBER, out1 => "DB440_MACHINE_ALARM_DECODING".GLOBAL_ALARMS_MACHINE.ALARM_DECODING)
      S_Coil( "DB440_MACHINE_ALARM_DECODING".ALARMS_UNIT_01.ST1_LOAD_UNLOAD.IS_SEOC_ALARMS )
   END_RUNG
   // the same network as SCL:
   // ENO of a box is taken as its EN; it also drops when the box reports an error
   IF NOT (NOT "DB1213_HOME_UNIT_01_STATION_1".SEQUENCE.TIME_EXCEEDED) THEN
       "DB440_MACHINE_ALARM_DECODING".GLOBAL_ALARMS_MACHINE.ALARM_DECODING := #FC_NUMBER;
       "DB440_MACHINE_ALARM_DECODING".ALARMS_UNIT_01.ST1_LOAD_UNLOAD.IS_SEOC_ALARMS := TRUE;
   END_IF;
END_REGION

REGION Network 20: GENERAL CONDITIONS HELP
   RUNG wire#powerrail
      Contact( "DB1213_HOME_UNIT_01_STATION_1".SEQUENCE.REQUEST )
      I_Contact( "DB1213_HOME_UNIT_01_STATION_1".SEQUENCE.GENERAL_CONDITIONS )
      I_Contact( "DB1213_HOME_UNIT_01_STATION_1".SEQUENCE.RUNNING )
      Coil( "DB1213_HOME_UNIT_01_STATION_1".SEQUENCE.GENERAL_CONDITIONS_HELP )
   END_RUNG
   // the same network as SCL:
   "DB1213_HOME_UNIT_01_STATION_1".SEQUENCE.GENERAL_CONDITIONS_HELP := "DB1213_HOME_UNIT_01_STATION_1".SEQUENCE.REQUEST AND NOT "DB1213_HOME_UNIT_01_STATION_1".SEQUENCE.GENERAL_CONDITIONS AND NOT "DB1213_HOME_UNIT_01_STATION_1".SEQUENCE.RUNNING;
END_REGION

REGION Network 21: INITIAL CONDITIONS HELP
   RUNG wire#powerrail
      Contact( "DB1213_HOME_UNIT_01_STATION_1".SEQUENCE.REQUEST )
      Contact( "DB1213_HOME_UNIT_01_STATION_1".SEQUENCE.GENERAL_CONDITIONS )
      I_Contact( "DB1213_HOME_UNIT_01_STATION_1".SEQUENCE.INITIAL_CONDITIONS )
      I_Contact( "DB1213_HOME_UNIT_01_STATION_1".SEQUENCE.RUNNING )
      Coil( "DB1213_HOME_UNIT_01_STATION_1".SEQUENCE.INITIAL_CONDITIONS_HELP )
   END_RUNG
   // the same network as SCL:
   "DB1213_HOME_UNIT_01_STATION_1".SEQUENCE.INITIAL_CONDITIONS_HELP := "DB1213_HOME_UNIT_01_STATION_1".SEQUENCE.REQUEST AND "DB1213_HOME_UNIT_01_STATION_1".SEQUENCE.GENERAL_CONDITIONS AND NOT "DB1213_HOME_UNIT_01_STATION_1".SEQUENCE.INITIAL_CONDITIONS AND NOT "DB1213_HOME_UNIT_01_STATION_1".SEQUENCE.RUNNING;
END_REGION

REGION Network 22: HMI STATUS
   RUNG wire#powerrail
      I_Contact( "DB1213_HOME_UNIT_01_STATION_1".SEQUENCE.RUNNING )
      Coil( "DB505_HMI_SetUp".Setup1.Movement_EndPos.movement231EndPosRight )
   END_RUNG
   // the same network as SCL:
   "DB505_HMI_SetUp".Setup1.Movement_EndPos.movement231EndPosRight := NOT "DB1213_HOME_UNIT_01_STATION_1".SEQUENCE.RUNNING;
END_REGION

REGION Network 23: HMI STATUS
   RUNG wire#powerrail
      Contact( "DB2001_MODES_GENERAL".GENERAL.SEMIAUTO_SELECTED )
      Contact( "DB1213_HOME_UNIT_01_STATION_1".SEQUENCE.GENERAL_CONDITIONS )
      Contact( "DB1213_HOME_UNIT_01_STATION_1".SEQUENCE.INITIAL_CONDITIONS )
      Coil( "DB505_HMI_SetUp".Setup1.Movement_Executability.movement231ExecutabilityRight )
   END_RUNG
   // the same network as SCL:
   "DB505_HMI_SetUp".Setup1.Movement_Executability.movement231ExecutabilityRight := "DB2001_MODES_GENERAL".GENERAL.SEMIAUTO_SELECTED AND "DB1213_HOME_UNIT_01_STATION_1".SEQUENCE.GENERAL_CONDITIONS AND "DB1213_HOME_UNIT_01_STATION_1".SEQUENCE.INITIAL_CONDITIONS;
END_REGION

REGION Network 24: HMI STATUS
   RUNG wire#powerrail
      Contact( "DB1213_HOME_UNIT_01_STATION_1".SEQUENCE.RUNNING )
      Contact( "M_0.5_SEC_2HZ" )
      Coil( "DB505_HMI_SetUp".Setup1.MovementActive.movement231ActiveRight )
   END_RUNG
   // the same network as SCL:
   "DB505_HMI_SetUp".Setup1.MovementActive.movement231ActiveRight := "DB1213_HOME_UNIT_01_STATION_1".SEQUENCE.RUNNING AND "M_0.5_SEC_2HZ";
END_REGION
END_FUNCTION
